// TIA Portal V18 export
TYPE "UDT_AHUsSustainedRequests"
// stored: IsFailsafeCompliant false
   STRUCT
      xNightCooling : Array[1..3] of Bool;
      xSustainedOnCooling : Array[1..3] of Bool;
      xSustainedOnHeating : Array[1..3] of Bool;
      xSusteinedOnIAQ : Array[1..3] of Bool;
      xSusteainedOnBuildingdP : Array[1..3] of Bool;
      cSummarySustTempRequest : Array[1..3] of Byte;
      xStartRequest : Array[1..3] of Bool;
      xBlockRequest : Array[1..3] of Bool;
   END_STRUCT;
END_TYPE
